PROGRAM MAIN
VAR
	my_real: REAL := 0.0;
END_VAR

END_PROGRAM

(* stored: Version 1.1.0.1, ProductVersion 3.1.0.36
   POU MAIN: Id {d2f6fade-e87b-4f9a-9ae6-16299feddd7a}, SpecialFunc None *)
